Staubli VAL3: moveC.pgx

public program moveC(point x_pInter (dimensions=1), point x_pLoc (dimensions=1), tool x_tTool (dimensions=1), mdesc x_mDesc (dimensions=1), num& x_nMoveID (dimensions=1), num& x_nError[] (dimensions=1))
// Perform a circular motion synchronized with a conveyor
  local num l_bLock
  local num l_bQuit
  local num l_nIdxInUse
  local string l_str
begin
  // This program executes a motion in tracking mode
  //
  // Input Param
  //  x_pInter  : Intermediate location of the circle
  //  x_pLoc    : Location to reach
  //  x_tTool   : Tool for motion
  //  x_nMoveID : ID of the movement on the motion stack
  //  x_mDesc   : Motion descriptor
  //
  // Output Param
  //  x_nError  : Error code
  //            = 0 : No error
  //            = 1 : No object ID selected
  //            = 3 : Bad conveyor number
  //
  //----------------------------------------------------------------
  //
  x_nError=0
  call whichObjectUsed(nCnvSynch,l_nIdxInUse,x_nError)
  if x_nError==0
    // Check if an object is in use (user must have invoked getNextID)
    if l_nIdxInUse!=-1
      tTool.trsf=position(x_tTool,flange)
      mTracking=x_mDesc
      if mTracking.blend==joint
        mTracking.blend=Cartesian
      endIf
      // Check robot type
      if bIsScara
        // Link locations to the mobile frame
        link(pInterTrack_RS,fMobileFrame[nMobFrameSync])
        pInterTrack_RS.trsf=position(x_pInter,fConveyor[nCnvSynch])
        pInterTrack_RS.config=x_pInter.config
        link(pTracking_RS,fMobileFrame[nMobFrameSync])
        pTracking_RS.trsf=position(x_pLoc,fConveyor[nCnvSynch])
        pTracking_RS.config=x_pLoc.config
        x_nMoveID=$movect(pInterTrack_RS,pTracking_RS,tTool,mTracking)
      else
        // Link locations to the mobile frame
        link(pInterTrack,fMobileFrame[nMobFrameSync])
        pInterTrack.trsf=position(x_pInter,fConveyor[nCnvSynch])
        pInterTrack.config=x_pInter.config
        link(pTracking,fMobileFrame[nMobFrameSync])
        pTracking.trsf=position(x_pLoc,fConveyor[nCnvSynch])
        pTracking.config=x_pLoc.config
        x_nMoveID=$movect(pInterTrack,pTracking,tTool,mTracking)
      endIf
      if bAnd(cfg:nLog,cfg:nLOGMOTION)==cfg:nLOGMOTION
        ? "MOT(moveC)>>Synchronised motion requested"
      endIf
    else
      if bAnd(cfg:nLog,cfg:nLOGMOTION)==cfg:nLOGMOTION
        ? "MOT(moveC)>>No object selected from queue"
      endIf
      x_nError=1
    endIf
  else
    if bAnd(cfg:nLog,cfg:nLOGMOTION)==cfg:nLOGMOTION
      ? "MOT(moveC)>>Invalid conveyor number: "+toString("",nCnvSynch)
    endIf
    x_nError=3
  endIf
end
